// TIA Portal V20 export
FUNCTION_BLOCK "Simulation_Actuator"   // FB110, LAD
// stored: Access Published, MemoryReserve 100, SetENOAutomatically false
   VAR_INPUT
      cmdHomePos : Bool;
      cmdWorkPos : Bool;
   END_VAR
   VAR_OUTPUT
      homePos : Bool;
      WorkPos : Bool;
   END_VAR
   VAR
      instTON { S7_SetPoint := 'True'} : Array[0..9] of TON_TIME;
   END_VAR
   VAR CONSTANT
      delayTime : Time := T#1s;
   END_VAR
BEGIN

REGION Network 1: Sylinder
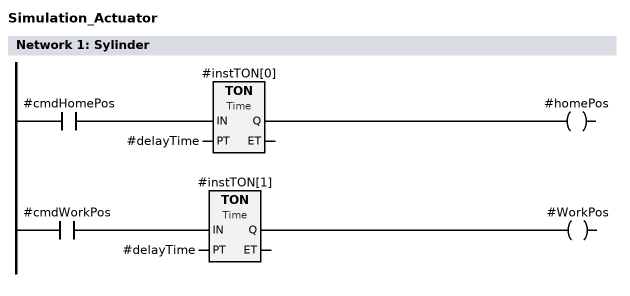
   RUNG wire#powerrail
      Contact( #cmdHomePos )
      { S7_Templates := "time_type := Time" } #instTON[0].TON(pt := #delayTime, et =>)
      Coil( #homePos )
   END_RUNG
   RUNG wire#powerrail
      Contact( #cmdWorkPos )
      { S7_Templates := "time_type := Time" } #instTON[1].TON(pt := #delayTime, et =>)
      Coil( #WorkPos )
   END_RUNG
   // the same network as SCL:
   #instTON[0].TON(IN := #cmdHomePos, PT := #delayTime);
   #homePos := #instTON[0].Q;
   #instTON[1].TON(IN := #cmdWorkPos, PT := #delayTime);
   #WorkPos := #instTON[1].Q;
END_REGION
END_FUNCTION_BLOCK
